{attribute 'analysis' := '-33'}
PROGRAM INTERNAL PRG_UnitTests
VAR
{IF defined (UNIT_TEST)}	
	fbJsonSerializerTests 	: FB_JsonSerializer_Tests;
	fbSnappyTests			: FB_Snappy_Tests;
{END_IF}
END_VAR

{IF defined (UNIT_TEST)}

TcUnit.RUN();

{END_IF}

END_PROGRAM

(* stored: Version 1.1.0.1, ProductVersion 3.1.4026.18
   POU PRG_UnitTests: Id {2224facc-781a-4d9f-985f-4e92aac79dd6}, SpecialFunc None *)
